// TIA Portal project "Lab2" (V15)

(* hardware
DEVICE "S71500/ET200MP station_1"  S7-1500 station
   slot 0: "Rail_0"  Rack  6ES7 590-1***0-0AA0
   slot 1: "PLC_1"  CPU 1511-1 PN  6ES7 511-1AK00-0AB0  V1.0
      slot 3: "CPU display_1"  6ES7591-1XA00-0AA0
   slot 2: "DI 16x24VDC HF_1"  DI 16x24VDC HF  6ES7 521-1BH00-0AB0  V1.0
   slot 3: "DQ 16x24VDC/0.5A ST_1"  DQ 16x24VDC/0.5A ST  6ES7 522-1BH00-0AB0  V1.0
   slot 4: "AI 8xU/I/RTD/TC ST_1"  AI 8xU/I/RTD/TC ST  6ES7 531-7KF00-0AB0  V2.0
*)

// ===== PLC "PLC_1"  CPU 1511-1 PN =====

VAR_GLOBAL   // PLC tag table "Default tag table"
   "K1_L" AT %I0.0 : Bool;
   "K1_R" AT %I0.1 : Bool;
   "K2_L" AT %I0.2 : Bool;
   "K2_R" AT %I0.3 : Bool;
   "K3_L" AT %I0.4 : Bool;
   "K3_R" AT %I0.5 : Bool;
   "K4_L" AT %I0.6 : Bool;
   "K4_R" AT %I0.7 : Bool;
   "K1_CL" AT %Q0.0 : Bool;
   "K1_CR" AT %Q0.1 : Bool;
   "K2_CL" AT %Q0.2 : Bool;
   "K2_CR" AT %Q0.3 : Bool;
   "K3_CL" AT %Q0.4 : Bool;
   "K4_CL" AT %Q0.6 : Bool;
   "K1_P" AT %IW2 : Word;
   "K3_P" AT %IW4 : Word;
END_VAR

DATA_BLOCK "Lab2_DB"   // DB1
{ S7_Optimized_Access := 'TRUE' }
VERSION : 0.1
   VAR
      State : Int;
      Done1 : Bool;
      Done2 : Bool;
      Done3 : Bool;
      Done4 : Bool;
      BeginWait : Bool;
      DoneWait : Bool;
      Set_Point_1 : Int;
      Set_Point_2 : Int;
      Set_Point_3 : Int;
      Set_Point_4 : Int;
      State6_Cnt : Int;
      State10_Cnt : Int;
      Discard1 : Bool;
      Discard2 : Bool;
   END_VAR
BEGIN
END_DATA_BLOCK

// folder: System blocks/Program resources

DATA_BLOCK "Lab2_Timer_DB"   // DB2
{ S7_Optimized_Access := 'TRUE' }
AUTHOR : Simatic
FAMILY : IEC
NAME : IEC_TMR
VERSION : 1.0
// stored: InstanceOfName IEC_TIMER
"IEC_TIMER"
BEGIN
END_DATA_BLOCK

// folder: (top level)

FUNCTION_BLOCK "MMC"   // FB1, LAD
{ S7_Optimized_Access := 'TRUE' }
VERSION : 0.1
   VAR_INPUT
      SP : Int;
   END_VAR
   VAR_OUTPUT
      D : Bool;
   END_VAR
   VAR
      aa : Int;
      IEC_Timer_0_Instance : TON_TIME;
   END_VAR
BEGIN

REGION Network 1
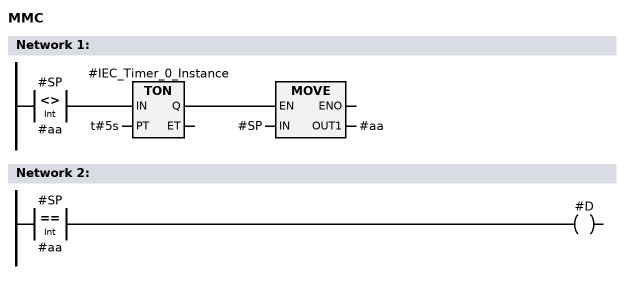
   #IEC_Timer_0_Instance(IN := #SP <> #aa, PT := t#5s);   // TON
   IF #IEC_Timer_0_Instance.Q THEN #aa := #SP; END_IF;
END_REGION

REGION Network 2
   RUNG wire#powerrail
      { S7_Templates := "SrcType := Int" } EQ_Contact(in1 := #SP, in2 := #aa)
      Coil( #D )
   END_RUNG
   // the same network as SCL:
   #D := #SP = #aa;
END_REGION
END_FUNCTION_BLOCK

FUNCTION "State_Await" : Void   // FC2, LAD
{ S7_Optimized_Access := 'TRUE' }
VERSION : 0.1
   VAR_TEMP
      All_Done : Bool;
   END_VAR
BEGIN

REGION Network 1
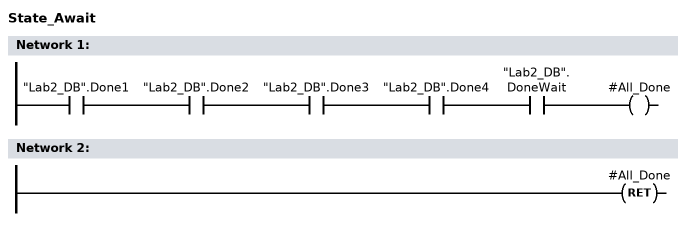
   RUNG wire#powerrail
      Contact( "Lab2_DB".Done1 )
      Contact( "Lab2_DB".Done2 )
      Contact( "Lab2_DB".Done3 )
      Contact( "Lab2_DB".Done4 )
      Contact( "Lab2_DB".DoneWait )
      Coil( #All_Done )
   END_RUNG
   // the same network as SCL:
   #All_Done := "Lab2_DB".Done1 AND "Lab2_DB".Done2 AND "Lab2_DB".Done3 AND "Lab2_DB".Done4 AND "Lab2_DB".DoneWait;
END_REGION

REGION Network 2
   ENO := #All_Done;
   RETURN;
END_REGION
END_FUNCTION

FUNCTION "Lab2_Motion_Control" : Void   // FC3, LAD
{ S7_Optimized_Access := 'TRUE' }
VERSION : 0.1
   VAR_INPUT
      Set_Point : Int;
      Sensor_Left : Bool;
      Sensor_Right : Bool;
      Sensor_Analog : Int;
   END_VAR
   VAR_OUTPUT
      Move_Left : Bool;
      Move_Right : Bool;
      Done : Bool;
   END_VAR
   VAR_TEMP
      Target_Value : Int;
      Current_Value : Int;
      Tmp_Diff : Int;
      Tmp_ADiff : Int;
   END_VAR
   VAR_TEMP   // added for the SCL form of the ladder/FBD networks
      _w1 : Bool;
   END_VAR
BEGIN

REGION Network 1
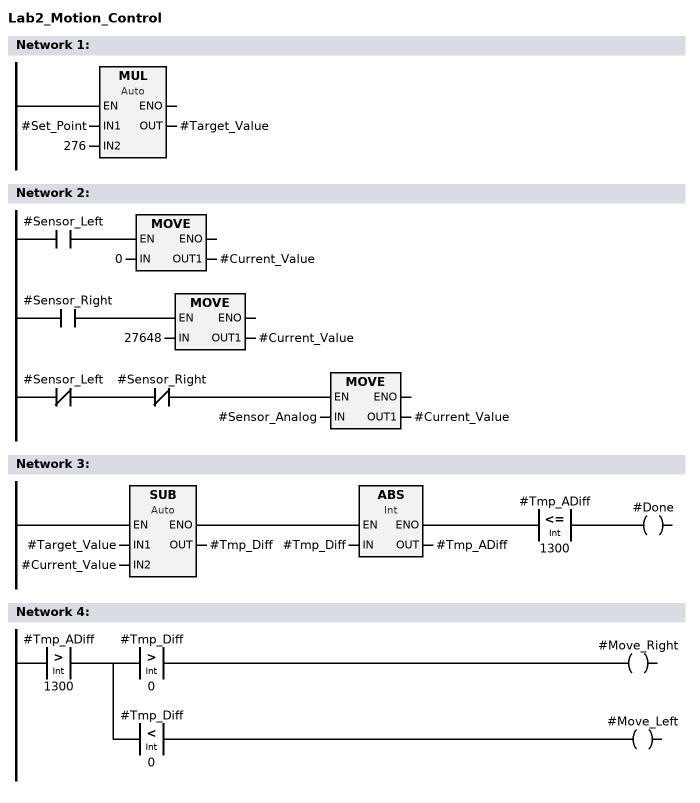
   RUNG wire#powerrail
      Mul(in1 := #Set_Point, in2 := 276, out => #Target_Value)
   END_RUNG
   // the same network as SCL:
   #Target_Value := #Set_Point * 276;
END_REGION

REGION Network 2
   RUNG wire#powerrail
      Contact( #Sensor_Left )
      Move(in := 0, out1 => #Current_Value)
   END_RUNG
   RUNG wire#powerrail
      Contact( #Sensor_Right )
      Move(in := 27648, out1 => #Current_Value)
   END_RUNG
   RUNG wire#powerrail
      I_Contact( #Sensor_Left )
      I_Contact( #Sensor_Right )
      Move(in := #Sensor_Analog, out1 => #Current_Value)
   END_RUNG
   // the same network as SCL:
   IF #Sensor_Left THEN #Current_Value := 0; END_IF;
   IF #Sensor_Right THEN #Current_Value := 27648; END_IF;
   IF NOT #Sensor_Left AND NOT #Sensor_Right THEN #Current_Value := #Sensor_Analog; END_IF;
END_REGION

REGION Network 3
   RUNG wire#powerrail
      Sub(in1 := #Target_Value, in2 := #Current_Value, out => #Tmp_Diff)
      { S7_Templates := "SrcType := Int" } Abs(in := #Tmp_Diff, out => #Tmp_ADiff)
      { S7_Templates := "SrcType := Int" } LE_Contact(in1 := #Tmp_ADiff, in2 := 1300)
      Coil( #Done )
   END_RUNG
   // the same network as SCL:
   #Tmp_Diff := #Target_Value - #Current_Value;
   #Tmp_ADiff := ABS(#Tmp_Diff);
   #Done := #Tmp_ADiff <= 1300;
END_REGION

REGION Network 4
   RUNG wire#powerrail
      { S7_Templates := "SrcType := Int" } GT_Contact(in1 := #Tmp_ADiff, in2 := 1300)
      wire#w1
      { S7_Templates := "SrcType := Int" } GT_Contact(in1 := #Tmp_Diff, in2 := 0)
      Coil( #Move_Right )
   END_RUNG
   RUNG wire#w1
      { S7_Templates := "SrcType := Int" } LT_Contact(in1 := #Tmp_Diff, in2 := 0)
      Coil( #Move_Left )
   END_RUNG
   // the same network as SCL:
   #_w1 := #Tmp_ADiff > 1300;
   #Move_Right := #_w1 AND (#Tmp_Diff > 0);
   #Move_Left := #_w1 AND (#Tmp_Diff < 0);
END_REGION
END_FUNCTION

ORGANIZATION_BLOCK "Main"   // OB1, LAD, ProgramCycle
TITLE = "Main Program Sweep (Cycle)"
{ S7_Optimized_Access := 'TRUE' }
VERSION : 0.1
   VAR_INPUT
      Initial_Call : Bool;   // Initial call of this OB
      Remanence : Bool;   // =True, if remanent data are available
   END_VAR
   VAR_TEMP   // added for the SCL form of the ladder/FBD networks
      _w1 : Bool;
      _w2 : Bool;
      _w3 : Bool;
   END_VAR
BEGIN

REGION Network 1
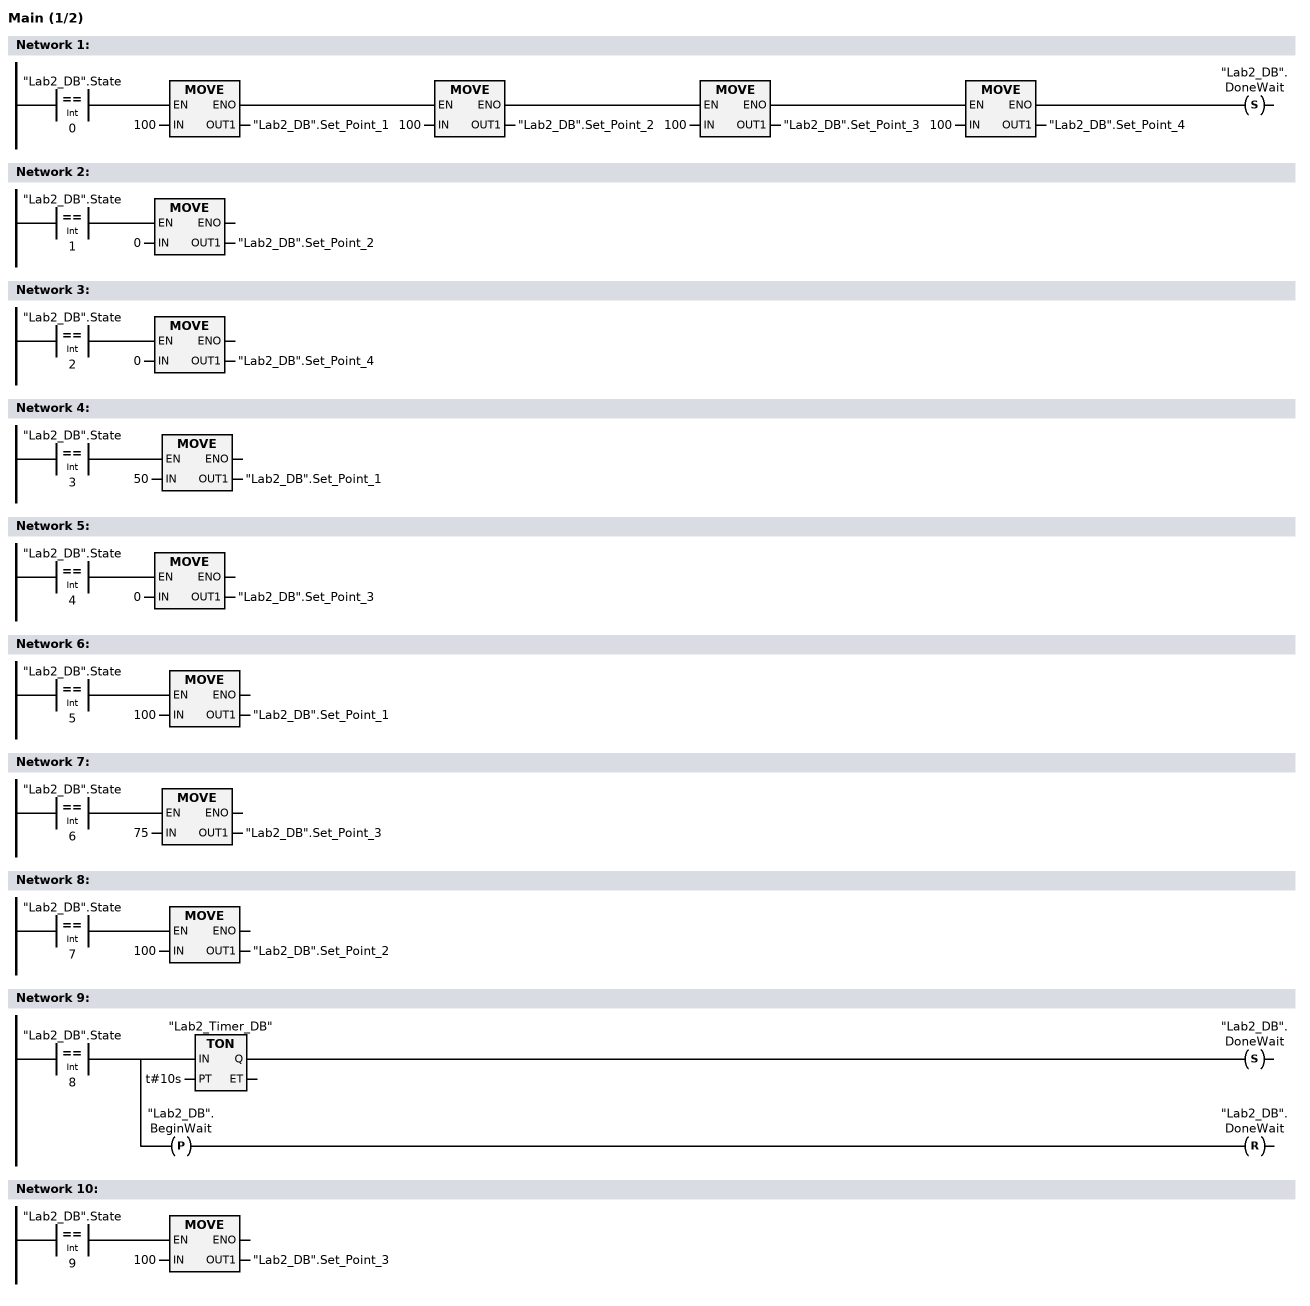
   RUNG wire#powerrail
      { S7_Templates := "SrcType := Int" } EQ_Contact(in1 := "Lab2_DB".State, in2 := 0)
      Move(in := 100, out1 => "Lab2_DB".Set_Point_1)
      Move(in := 100, out1 => "Lab2_DB".Set_Point_2)
      Move(in := 100, out1 => "Lab2_DB".Set_Point_3)
      Move(in := 100, out1 => "Lab2_DB".Set_Point_4)
      S_Coil( "Lab2_DB".DoneWait )
   END_RUNG
   // the same network as SCL:
   IF "Lab2_DB".State = 0 THEN
       "Lab2_DB".Set_Point_1 := 100;
       "Lab2_DB".Set_Point_2 := 100;
       "Lab2_DB".Set_Point_3 := 100;
       "Lab2_DB".Set_Point_4 := 100;
       "Lab2_DB".DoneWait := TRUE;
   END_IF;
END_REGION

REGION Network 2
   RUNG wire#powerrail
      { S7_Templates := "SrcType := Int" } EQ_Contact(in1 := "Lab2_DB".State, in2 := 1)
      Move(in := 0, out1 => "Lab2_DB".Set_Point_2)
   END_RUNG
   // the same network as SCL:
   IF "Lab2_DB".State = 1 THEN "Lab2_DB".Set_Point_2 := 0; END_IF;
END_REGION

REGION Network 3
   RUNG wire#powerrail
      { S7_Templates := "SrcType := Int" } EQ_Contact(in1 := "Lab2_DB".State, in2 := 2)
      Move(in := 0, out1 => "Lab2_DB".Set_Point_4)
   END_RUNG
   // the same network as SCL:
   IF "Lab2_DB".State = 2 THEN "Lab2_DB".Set_Point_4 := 0; END_IF;
END_REGION

REGION Network 4
   RUNG wire#powerrail
      { S7_Templates := "SrcType := Int" } EQ_Contact(in1 := "Lab2_DB".State, in2 := 3)
      Move(in := 50, out1 => "Lab2_DB".Set_Point_1)
   END_RUNG
   // the same network as SCL:
   IF "Lab2_DB".State = 3 THEN "Lab2_DB".Set_Point_1 := 50; END_IF;
END_REGION

REGION Network 5
   RUNG wire#powerrail
      { S7_Templates := "SrcType := Int" } EQ_Contact(in1 := "Lab2_DB".State, in2 := 4)
      Move(in := 0, out1 => "Lab2_DB".Set_Point_3)
   END_RUNG
   // the same network as SCL:
   IF "Lab2_DB".State = 4 THEN "Lab2_DB".Set_Point_3 := 0; END_IF;
END_REGION

REGION Network 6
   RUNG wire#powerrail
      { S7_Templates := "SrcType := Int" } EQ_Contact(in1 := "Lab2_DB".State, in2 := 5)
      Move(in := 100, out1 => "Lab2_DB".Set_Point_1)
   END_RUNG
   // the same network as SCL:
   IF "Lab2_DB".State = 5 THEN "Lab2_DB".Set_Point_1 := 100; END_IF;
END_REGION

REGION Network 7
   RUNG wire#powerrail
      { S7_Templates := "SrcType := Int" } EQ_Contact(in1 := "Lab2_DB".State, in2 := 6)
      Move(in := 75, out1 => "Lab2_DB".Set_Point_3)
   END_RUNG
   // the same network as SCL:
   IF "Lab2_DB".State = 6 THEN "Lab2_DB".Set_Point_3 := 75; END_IF;
END_REGION

REGION Network 8
   RUNG wire#powerrail
      { S7_Templates := "SrcType := Int" } EQ_Contact(in1 := "Lab2_DB".State, in2 := 7)
      Move(in := 100, out1 => "Lab2_DB".Set_Point_2)
   END_RUNG
   // the same network as SCL:
   IF "Lab2_DB".State = 7 THEN "Lab2_DB".Set_Point_2 := 100; END_IF;
END_REGION

REGION Network 9
   #_w1 := "Lab2_DB".State = 8;
   "Lab2_Timer_DB".TON(IN := #_w1, PT := t#10s);
   IF "Lab2_Timer_DB".Q THEN "Lab2_DB".DoneWait := TRUE; END_IF;
   #_w2 := #_w1 AND NOT "Lab2_DB".BeginWait;   // rising edge
   "Lab2_DB".BeginWait := #_w1;
   IF #_w2 THEN "Lab2_DB".DoneWait := FALSE; END_IF;
END_REGION

REGION Network 10
   RUNG wire#powerrail
      { S7_Templates := "SrcType := Int" } EQ_Contact(in1 := "Lab2_DB".State, in2 := 9)
      Move(in := 100, out1 => "Lab2_DB".Set_Point_3)
   END_RUNG
   // the same network as SCL:
   IF "Lab2_DB".State = 9 THEN "Lab2_DB".Set_Point_3 := 100; END_IF;
END_REGION

REGION Network 11
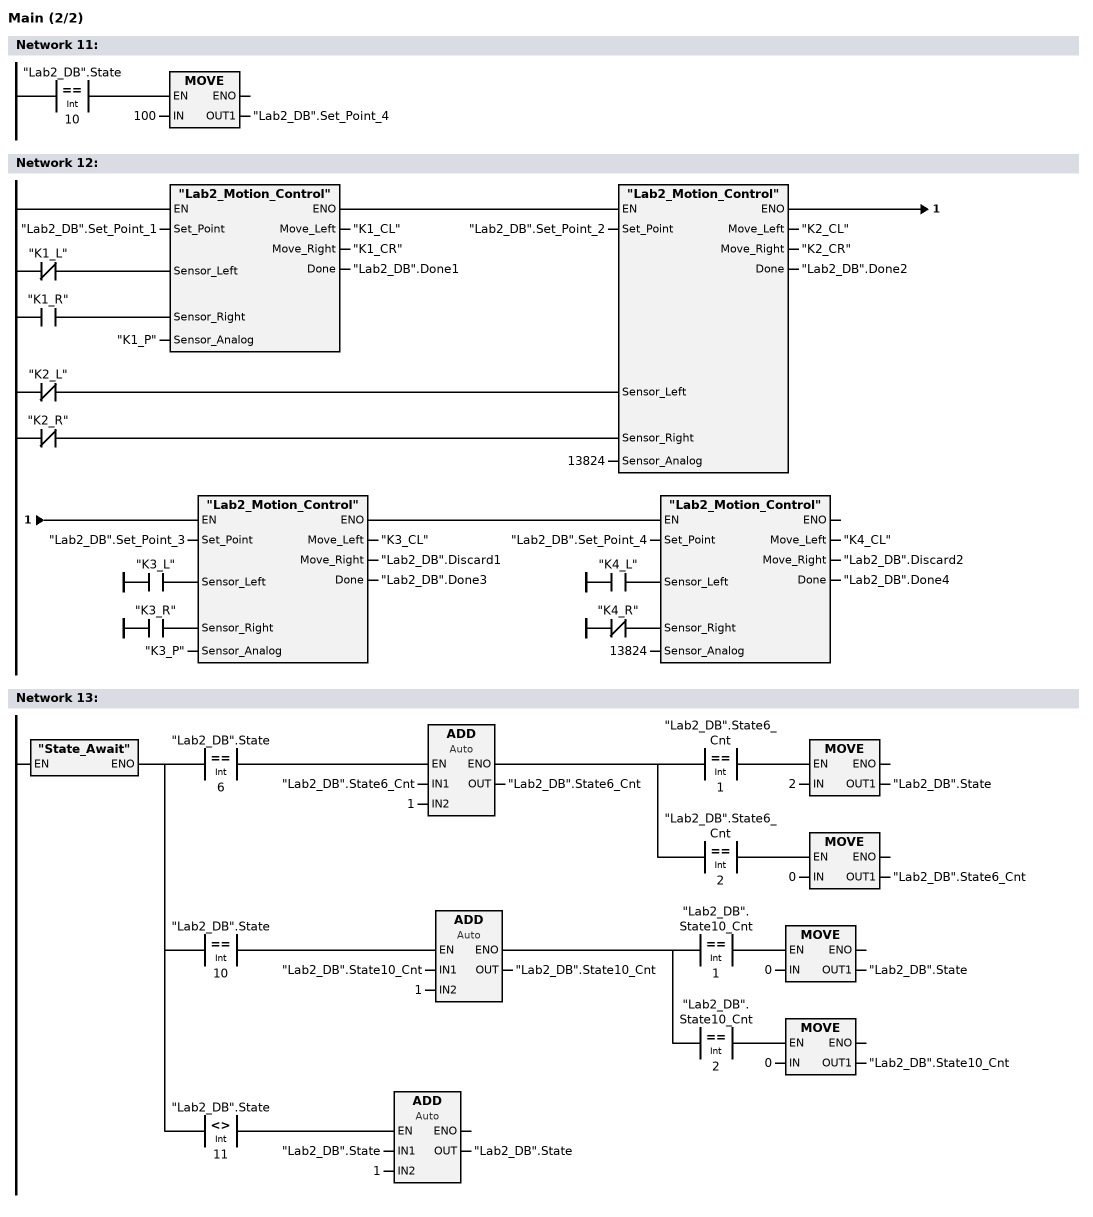
   RUNG wire#powerrail
      { S7_Templates := "SrcType := Int" } EQ_Contact(in1 := "Lab2_DB".State, in2 := 10)
      Move(in := 100, out1 => "Lab2_DB".Set_Point_4)
   END_RUNG
   // the same network as SCL:
   IF "Lab2_DB".State = 10 THEN "Lab2_DB".Set_Point_4 := 100; END_IF;
END_REGION

REGION Network 12
   RUNG wire#powerrail
      "Lab2_Motion_Control"(Sensor_Left := wire#w1, Sensor_Right := wire#w2, Set_Point := "Lab2_DB".Set_Point_1, Sensor_Analog := "K1_P", Move_Left => "K1_CL", Move_Right => "K1_CR", Done => "Lab2_DB".Done1)
      "Lab2_Motion_Control"(Sensor_Left := wire#w3, Sensor_Right := wire#w4, Set_Point := "Lab2_DB".Set_Point_2, Sensor_Analog := 13824, Move_Left => "K2_CL", Move_Right => "K2_CR", Done => "Lab2_DB".Done2)
      "Lab2_Motion_Control"(Sensor_Left := wire#w5, Sensor_Right := wire#w6, Set_Point := "Lab2_DB".Set_Point_3, Sensor_Analog := "K3_P", Move_Left => "K3_CL", Move_Right => "Lab2_DB".Discard1, Done => "Lab2_DB".Done3)
      "Lab2_Motion_Control"(Sensor_Left := wire#w7, Sensor_Right := wire#w8, Set_Point := "Lab2_DB".Set_Point_4, Sensor_Analog := 13824, Move_Left => "K4_CL", Move_Right => "Lab2_DB".Discard2, Done => "Lab2_DB".Done4)
   END_RUNG
   RUNG wire#powerrail
      I_Contact( "K1_L" )
   END_RUNG wire#w1
   RUNG wire#powerrail
      Contact( "K1_R" )
   END_RUNG wire#w2
   RUNG wire#powerrail
      I_Contact( "K2_L" )
   END_RUNG wire#w3
   RUNG wire#powerrail
      I_Contact( "K2_R" )
   END_RUNG wire#w4
   RUNG wire#powerrail
      Contact( "K3_L" )
   END_RUNG wire#w5
   RUNG wire#powerrail
      Contact( "K3_R" )
   END_RUNG wire#w6
   RUNG wire#powerrail
      Contact( "K4_L" )
   END_RUNG wire#w7
   RUNG wire#powerrail
      I_Contact( "K4_R" )
   END_RUNG wire#w8
   // the same network as SCL:
   "Lab2_Motion_Control"(Set_Point := "Lab2_DB".Set_Point_1,
                         Sensor_Left := NOT "K1_L",
                         Sensor_Right := "K1_R",
                         Sensor_Analog := "K1_P",
                         Move_Left => "K1_CL",
                         Move_Right => "K1_CR",
                         Done => "Lab2_DB".Done1,
                         ENO => #_w1);
   "Lab2_Motion_Control"(EN := #_w1,
                         Set_Point := "Lab2_DB".Set_Point_2,
                         Sensor_Left := NOT "K2_L",
                         Sensor_Right := NOT "K2_R",
                         Sensor_Analog := 13824,
                         Move_Left => "K2_CL",
                         Move_Right => "K2_CR",
                         Done => "Lab2_DB".Done2,
                         ENO => #_w2);
   "Lab2_Motion_Control"(EN := #_w2,
                         Set_Point := "Lab2_DB".Set_Point_3,
                         Sensor_Left := "K3_L",
                         Sensor_Right := "K3_R",
                         Sensor_Analog := "K3_P",
                         Move_Left => "K3_CL",
                         Move_Right => "Lab2_DB".Discard1,
                         Done => "Lab2_DB".Done3,
                         ENO => #_w3);
   IF #_w3 THEN
       "Lab2_Motion_Control"(Set_Point := "Lab2_DB".Set_Point_4,
                             Sensor_Left := "K4_L",
                             Sensor_Right := NOT "K4_R",
                             Sensor_Analog := 13824,
                             Move_Left => "K4_CL",
                             Move_Right => "Lab2_DB".Discard2,
                             Done => "Lab2_DB".Done4);
   END_IF;
END_REGION

REGION Network 13
   RUNG wire#powerrail
      "State_Await"()
      wire#w1
      { S7_Templates := "SrcType := Int" } EQ_Contact(in1 := "Lab2_DB".State, in2 := 6)
      Add(in1 := "Lab2_DB".State6_Cnt, in2 := 1, out => "Lab2_DB".State6_Cnt)
      wire#w2
      { S7_Templates := "SrcType := Int" } EQ_Contact(in1 := "Lab2_DB".State6_Cnt, in2 := 1)
      Move(in := 2, out1 => "Lab2_DB".State)
   END_RUNG
   RUNG wire#w2
      { S7_Templates := "SrcType := Int" } EQ_Contact(in1 := "Lab2_DB".State6_Cnt, in2 := 2)
      Move(in := 0, out1 => "Lab2_DB".State6_Cnt)
   END_RUNG
   RUNG wire#w1
      { S7_Templates := "SrcType := Int" } EQ_Contact(in1 := "Lab2_DB".State, in2 := 10)
      Add(in1 := "Lab2_DB".State10_Cnt, in2 := 1, out => "Lab2_DB".State10_Cnt)
      wire#w3
      { S7_Templates := "SrcType := Int" } EQ_Contact(in1 := "Lab2_DB".State10_Cnt, in2 := 1)
      Move(in := 0, out1 => "Lab2_DB".State)
   END_RUNG
   RUNG wire#w3
      { S7_Templates := "SrcType := Int" } EQ_Contact(in1 := "Lab2_DB".State10_Cnt, in2 := 2)
      Move(in := 0, out1 => "Lab2_DB".State10_Cnt)
   END_RUNG
   RUNG wire#w1
      { S7_Templates := "SrcType := Int" } NE_Contact(in1 := "Lab2_DB".State, in2 := 11)
      Add(in1 := "Lab2_DB".State, in2 := 1, out => "Lab2_DB".State)
   END_RUNG
   // the same network as SCL:
   "State_Await"(ENO => #_w1);
   #_w2 := #_w1 AND ("Lab2_DB".State = 6);
   IF #_w2 THEN "Lab2_DB".State6_Cnt := "Lab2_DB".State6_Cnt + 1; END_IF;
   IF #_w2 AND ("Lab2_DB".State6_Cnt = 1) THEN "Lab2_DB".State := 2; END_IF;
   IF #_w2 AND ("Lab2_DB".State6_Cnt = 2) THEN "Lab2_DB".State6_Cnt := 0; END_IF;
   #_w3 := #_w1 AND ("Lab2_DB".State = 10);
   IF #_w3 THEN "Lab2_DB".State10_Cnt := "Lab2_DB".State10_Cnt + 1; END_IF;
   IF #_w3 AND ("Lab2_DB".State10_Cnt = 1) THEN "Lab2_DB".State := 0; END_IF;
   IF #_w3 AND ("Lab2_DB".State10_Cnt = 2) THEN "Lab2_DB".State10_Cnt := 0; END_IF;
   IF #_w1 AND ("Lab2_DB".State <> 11) THEN "Lab2_DB".State := "Lab2_DB".State + 1; END_IF;
END_REGION
END_ORGANIZATION_BLOCK